INTERFACE I_XtsTrack

PROPERTY MyOTCID : OTCID
GET
END_GET
SET
END_SET
END_PROPERTY

PROPERTY TrackLength : MC_Lreal
GET
END_GET
END_PROPERTY

END_INTERFACE

(* stored: Version 1.1.0.1
   Itf I_XtsTrack: Id {b580e084-f2aa-4b9e-b34b-5773df679de5}
   Property MyOTCID: Id {8be67bfb-cfe2-4d62-98cc-25000c035505}
   Get Get: Id {4e95c9bb-aa4d-4ade-9bfa-d3c230375802}
   Set Set: Id {5a69d026-ba0e-42f2-ad56-82e6069370de}
   Property TrackLength: Id {d09b154e-641d-4452-b45a-353375f2a798}
   Get Get: Id {227be027-fd95-4a28-b451-be32068fa3af} *)
